LIN {X 0,Y 69.848,Z 476.675,A -85,B 0,C 180,E1 -28499.796,E2 -28499.796} C_VEL
LIN {X 0,Y 67.103,Z 478.987,A -85,B 0,C 180,E1 -28505.233,E2 -28505.233} C_VEL
LIN {X 0,Y 64.997,Z 480.714,A -85,B 0,C 180,E1 -28511.072,E2 -28511.072} C_VEL
LIN {X 0,Y 63.489,Z 481.949,A -85,B 0,C 180,E1 -28517.21,E2 -28517.21} C_VEL
LIN {X 0,Y 62.689,Z 482.712,A -85,B 0,C 180,E1 -28523.563,E2 -28523.563} C_VEL
LIN {X 0,Y 62.51,Z 483,A -85,B 0,C 180,E1 -28530,E2 -28530} C_VEL
LIN {X 0,Y 62.687,Z 482.698,A -85,B 0,C 180,E1 -28536.437,E2 -28536.437} C_VEL
LIN {X 0,Y 63.483,Z 481.907,A -85,B 0,C 180,E1 -28542.792,E2 -28542.792} C_VEL
LIN {X 0,Y 64.985,Z 480.644,A -85,B 0,C 180,E1 -28548.931,E2 -28548.931} C_VEL
LIN {X 0,Y 68.386,Z 477.737,A -85,B 0,C 180,E1 -28557.546,E2 -28557.546} C_VEL
LIN {X 0,Y 71.407,Z 475.084,A -85,B 0,C 180,E1 -28562.773,E2 -28562.773} C_VEL
LIN {X 0,Y 76.916,Z 469.904,A -85,B 0,C 180,E1 -28569.761,E2 -28569.761} C_VEL
LIN {X 0,Y 83.46,Z 463.065,A -85,B 0,C 180,E1 -28575.705,E2 -28575.705} C_VEL
LIN {X 0,Y 89.457,Z 455.594,A -85,B 0,C 180,E1 -28579.993,E2 -28579.993} C_VEL
LIN {X 0,Y 94.61,Z 448.222,A -85,B 0,C 180,E1 -28582.99,E2 -28582.99} C_VEL
LIN {X 0,Y 99.158,Z 440.542,A -85,B 0,C 180,E1 -28585.32,E2 -28585.32} C_VEL
LIN {X 0,Y 103.34,Z 431.965,A -85,B 0,C 180,E1 -28587.308,E2 -28587.308} C_VEL
LIN {X 0,Y 107.288,Z 421.966,A -85,B 0,C 180,E1 -28588.97,E2 -28588.97} C_VEL
LIN {X 0,Y 110.604,Z 410.25,A -85,B 0,C 180,E1 -28590.22,E2 -28590.22} C_VEL
LIN {X 0,Y 112.44,Z 400.537,A -85,B 0,C 180,E1 -28590.874,E2 -28590.874} C_VEL
LIN {X 0,Y 112.912,Z 396.513,A -85,B 0,C 180,E1 -28591.157,E2 -28591.157} C_VEL
LIN {X 0,Y 109.721,Z 389.352,A -85,B 0,C 180,E1 -28595.466,E2 -28595.466} C_VEL
LIN {X 0,Y 107.221,Z 384.494,A -85,B 0,C 180,E1 -28599.466,E2 -28599.466} C_VEL
LIN {X 0,Y 105.6,Z 381.525,A -85,B 0,C 180,E1 -28602.605,E2 -28602.605} C_VEL
LIN {X 0,Y 103.774,Z 378.179,A -85,B 0,C 180,E1 -28607.159,E2 -28607.159} C_VEL
LIN {X 0,Y 102.189,Z 375.125,A -85,B 0,C 180,E1 -28613.584,E2 -28613.584} C_VEL
LIN {X 0,Y 101.944,Z 373.871,A -85,B 0,C 180,E1 -28616.047,E2 -28616.047} C_VEL
LIN {X 0,Y 101.743,Z 373.505,A -85,B 0,C 180,E1 -28620,E2 -28620} C_VEL
LIN {X 0,Y 102.017,Z 374.037,A -85,B 0,C 180,E1 -28624.693,E2 -28624.693} C_VEL
LIN {X 0,Y 103.212,Z 377.51,A -85,B 0,C 180,E1 -28631.209,E2 -28631.209} C_VEL
LIN {X 0,Y 104.184,Z 378.885,A -85,B 0,C 180,E1 -28634.039,E2 -28634.039} C_VEL
LIN {X 0,Y 106.507,Z 383.167,A -85,B 0,C 180,E1 -28639.265,E2 -28639.265} C_VEL
LIN {X 0,Y 108.728,Z 387.363,A -85,B 0,C 180,E1 -28643.08,E2 -28643.08} C_VEL
LIN {X 0,Y 111.51,Z 393.241,A -85,B 0,C 180,E1 -28647.064,E2 -28647.064} C_VEL
LIN {X 0,Y 112.912,Z 396.627,A -85,B 0,C 180,E1 -28648.909,E2 -28648.909} C_VEL
LIN {X 0,Y 111.228,Z 407.408,A -85,B 0,C 180,E1 -28649.608,E2 -28649.608} C_VEL
LIN {X 0,Y 111.11,Z 407.875,A -85,B 0,C 180,E1 -28649.629,E2 -28649.629} C_VEL
LIN {X 0,Y 108.536,Z 415.532,A -85,B 0,C 180,E1 -28649.681,E2 -28649.681} C_VEL
LIN {X 0,Y 105.062,Z 422.853,A -85,B 0,C 180,E1 -28649.456,E2 -28649.456} C_VEL
LIN {X 0,Y 100.321,Z 431.414,A -85,B 0,C 180,E1 -28649.539,E2 -28649.539} C_VEL
LIN {X 0,Y 97.661,Z 436.251,A -85,B 0,C 180,E1 -28650.185,E2 -28650.185} C_VEL
LIN {X 0,Y 91.957,Z 446.132,A -85,B 0,C 180,E1 -28652.788,E2 -28652.788} C_VEL
LIN {X 0,Y 86.43,Z 453.852,A -85,B 0,C 180,E1 -28655.598,E2 -28655.598} C_VEL
LIN {X 0,Y 81.208,Z 460.199,A -85,B 0,C 180,E1 -28658.843,E2 -28658.843} C_VEL
LIN {X 0,Y 76.245,Z 465.475,A -85,B 0,C 180,E1 -28662.49,E2 -28662.49} C_VEL
LIN {X 0,Y 71.621,Z 469.88,A -85,B 0,C 180,E1 -28666.617,E2 -28666.617} C_VEL
LIN {X 0,Y 65.574,Z 475.065,A -85,B 0,C 180,E1 -28673.882,E2 -28673.882} C_VEL
LIN {X 0,Y 62.209,Z 477.722,A -85,B 0,C 180,E1 -28679.445,E2 -28679.445} C_VEL
LIN {X 0,Y 58.304,Z 480.634,A -85,B 0,C 180,E1 -28688.801,E2 -28688.801} C_VEL
LIN {X 0,Y 56.597,Z 481.901,A -85,B 0,C 180,E1 -28695.62,E2 -28695.62} C_VEL
LIN {X 0,Y 55.633,Z 482.696,A -85,B 0,C 180,E1 -28702.743,E2 -28702.743} C_VEL
LIN {X 0,Y 55.414,Z 482.999,A -85,B 0,C 180,E1 -28710,E2 -28710} C_VEL
LIN {X 0,Y 55.633,Z 482.714,A -85,B 0,C 180,E1 -28717.257,E2 -28717.257} C_VEL
LIN {X 0,Y 56.596,Z 481.955,A -85,B 0,C 180,E1 -28724.38,E2 -28724.38} C_VEL
LIN {X 0,Y 58.299,Z 480.725,A -85,B 0,C 180,E1 -28731.201,E2 -28731.201} C_VEL
LIN {X 0,Y 62.166,Z 477.851,A -85,B 0,C 180,E1 -28740.579,E2 -28740.579} C_VEL
LIN {X 0,Y 65.535,Z 475.234,A -85,B 0,C 180,E1 -28746.143,E2 -28746.143} C_VEL
LIN {X 0,Y 71.592,Z 470.095,A -85,B 0,C 180,E1 -28753.405,E2 -28753.405} C_VEL
LIN {X 0,Y 77.406,Z 464.567,A -85,B 0,C 180,E1 -28758.507,E2 -28758.507} C_VEL
LIN {X 0,Y 83.747,Z 457.615,A -85,B 0,C 180,E1 -28762.865,E2 -28762.865} C_VEL
LIN {X 0,Y 89.827,Z 449.637,A -85,B 0,C 180,E1 -28766.23,E2 -28766.23} C_VEL
LIN {X 0,Y 94.868,Z 441.786,A -85,B 0,C 180,E1 -28768.624,E2 -28768.624} C_VEL
LIN {X 0,Y 98.991,Z 434.053,A -85,B 0,C 180,E1 -28770.422,E2 -28770.422} C_VEL
LIN {X 0,Y 102.605,Z 425.802,A -85,B 0,C 180,E1 -28771.868,E2 -28771.868} C_VEL
LIN {X 0,Y 105.581,Z 417.212,A -85,B 0,C 180,E1 -28772.998,E2 -28772.998} C_VEL
LIN {X 0,Y 108.054,Z 407.867,A -85,B 0,C 180,E1 -28773.822,E2 -28773.822} C_VEL
LIN {X 0,Y 109.442,Z 400.033,A -85,B 0,C 180,E1 -28774.344,E2 -28774.344} C_VEL
LIN {X 0,Y 107.116,Z 394.028,A -85,B 0,C 180,E1 -28778.389,E2 -28778.389} C_VEL
LIN {X 0,Y 105.229,Z 390.11,A -85,B 0,C 180,E1 -28781.975,E2 -28781.975} C_VEL
LIN {X 0,Y 104.07,Z 387.868,A -85,B 0,C 180,E1 -28784.61,E2 -28784.61} C_VEL
LIN {X 0,Y 102.85,Z 385.178,A -85,B 0,C 180,E1 -28788.17,E2 -28788.17} C_VEL
LIN {X 0,Y 101.381,Z 381.825,A -85,B 0,C 180,E1 -28795.527,E2 -28795.527} C_VEL
LIN {X 0,Y 101.306,Z 381.029,A -85,B 0,C 180,E1 -28797.017,E2 -28797.017} C_VEL
LIN {X 0,Y 101.207,Z 380.698,A -85,B 0,C 180,E1 -28800,E2 -28800} C_VEL
LIN {X 0,Y 101.327,Z 381.227,A -85,B 0,C 180,E1 -28803.479,E2 -28803.479} C_VEL
LIN {X 0,Y 102.534,Z 384.8,A -85,B 0,C 180,E1 -28810.864,E2 -28810.864} C_VEL
LIN {X 0,Y 103.118,Z 385.874,A -85,B 0,C 180,E1 -28812.781,E2 -28812.781} C_VEL
LIN {X 0,Y 104.964,Z 389.588,A -85,B 0,C 180,E1 -28817.504,E2 -28817.504} C_VEL
LIN {X 0,Y 106.974,Z 393.735,A -85,B 0,C 180,E1 -28821.411,E2 -28821.411} C_VEL
LIN {X 0,Y 109.14,Z 399.137,A -85,B 0,C 180,E1 -28825.182,E2 -28825.182} C_VEL
LIN {X 0,Y 109.44,Z 400.029,A -85,B 0,C 180,E1 -28825.698,E2 -28825.698} C_VEL
LIN {X 0,Y 108.079,Z 407.829,A -85,B 0,C 180,E1 -28826.237,E2 -28826.237} C_VEL
LIN {X 0,Y 105.622,Z 417.18,A -85,B 0,C 180,E1 -28827.076,E2 -28827.076} C_VEL
LIN {X 0,Y 102.616,Z 425.721,A -85,B 0,C 180,E1 -28828.144,E2 -28828.144} C_VEL
LIN {X 0,Y 98.992,Z 433.988,A -85,B 0,C 180,E1 -28829.579,E2 -28829.579} C_VEL
LIN {X 0,Y 94.079,Z 443.081,A -85,B 0,C 180,E1 -28831.716,E2 -28831.716} C_VEL
LIN {X 0,Y 87.769,Z 452.48,A -85,B 0,C 180,E1 -28834.842,E2 -28834.842} C_VEL
LIN {X 0,Y 82.475,Z 459.063,A -85,B 0,C 180,E1 -28837.982,E2 -28837.982} C_VEL
LIN {X 0,Y 77.428,Z 464.54,A -85,B 0,C 180,E1 -28841.512,E2 -28841.512} C_VEL
LIN {X 0,Y 71.605,Z 470.073,A -85,B 0,C 180,E1 -28846.605,E2 -28846.605} C_VEL
LIN {X 0,Y 65.542,Z 475.216,A -85,B 0,C 180,E1 -28853.861,E2 -28853.861} C_VEL
LIN {X 0,Y 60.733,Z 478.988,A -85,B 0,C 180,E1 -28862.428,E2 -28862.428} C_VEL
LIN {X 0,Y 58.308,Z 480.715,A -85,B 0,C 180,E1 -28868.802,E2 -28868.802} C_VEL
LIN {X 0,Y 56.6,Z 481.949,A -85,B 0,C 180,E1 -28875.621,E2 -28875.621} C_VEL
LIN {X 0,Y 55.633,Z 482.712,A -85,B 0,C 180,E1 -28882.743,E2 -28882.743} C_VEL
LIN {X 0,Y 55.412,Z 483,A -85,B 0,C 180,E1 -28890,E2 -28890} C_VEL
LIN {X 0,Y 55.631,Z 482.698,A -85,B 0,C 180,E1 -28897.258,E2 -28897.258} C_VEL
LIN {X 0,Y 56.594,Z 481.906,A -85,B 0,C 180,E1 -28904.38,E2 -28904.38} C_VEL
LIN {X 0,Y 58.299,Z 480.644,A -85,B 0,C 180,E1 -28911.201,E2 -28911.201} C_VEL
LIN {X 0,Y 62.174,Z 477.736,A -85,B 0,C 180,E1 -28920.575,E2 -28920.575} C_VEL
LIN {X 0,Y 65.537,Z 475.083,A -85,B 0,C 180,E1 -28926.142,E2 -28926.142} C_VEL
LIN {X 0,Y 71.604,Z 469.903,A -85,B 0,C 180,E1 -28933.396,E2 -28933.396} C_VEL
LIN {X 0,Y 78.672,Z 463.063,A -85,B 0,C 180,E1 -28939.403,E2 -28939.403} C_VEL
LIN {X 0,Y 85.067,Z 455.591,A -85,B 0,C 180,E1 -28943.658,E2 -28943.658} C_VEL
LIN {X 0,Y 90.522,Z 448.219,A -85,B 0,C 180,E1 -28946.574,E2 -28946.574} C_VEL
LIN {X 0,Y 94.728,Z 441.531,A -85,B 0,C 180,E1 -28948.573,E2 -28948.573} C_VEL
LIN {X 0,Y 98.974,Z 433.461,A -85,B 0,C 180,E1 -28950.439,E2 -28950.439} C_VEL
LIN {X 0,Y 102.601,Z 425.063,A -85,B 0,C 180,E1 -28951.872,E2 -28951.872} C_VEL
LIN {X 0,Y 105.779,Z 415.77,A -85,B 0,C 180,E1 -28953,E2 -28953} C_VEL
LIN {X 0,Y 108.637,Z 404.172,A -85,B 0,C 180,E1 -28953.921,E2 -28953.921} C_VEL
LIN {X 0,Y 109.195,Z 399.767,A -85,B 0,C 180,E1 -28954.249,E2 -28954.249} C_VEL
LIN {X 0,Y 106.787,Z 393.629,A -85,B 0,C 180,E1 -28958.399,E2 -28958.399} C_VEL
LIN {X 0,Y 104.405,Z 388.609,A -85,B 0,C 180,E1 -28963.109,E2 -28963.109} C_VEL
LIN {X 0,Y 102.537,Z 384.948,A -85,B 0,C 180,E1 -28968.134,E2 -28968.134} C_VEL
LIN {X 0,Y 101.136,Z 381.751,A -85,B 0,C 180,E1 -28974.892,E2 -28974.892} C_VEL
LIN {X 0,Y 100.984,Z 380.826,A -85,B 0,C 180,E1 -28977.008,E2 -28977.008} C_VEL
LIN {X 0,Y 100.877,Z 380.562,A -85,B 0,C 180,E1 -28980,E2 -28980} C_VEL
LIN {X 0,Y 101.06,Z 381.043,A -85,B 0,C 180,E1 -28983.988,E2 -28983.988} C_VEL
LIN {X 0,Y 102.175,Z 384.511,A -85,B 0,C 180,E1 -28990.741,E2 -28990.741} C_VEL
LIN {X 0,Y 102.8,Z 385.479,A -85,B 0,C 180,E1 -28992.752,E2 -28992.752} C_VEL
LIN {X 0,Y 104.924,Z 389.79,A -85,B 0,C 180,E1 -28998.101,E2 -28998.101} C_VEL
LIN {X 0,Y 107.067,Z 394.284,A -85,B 0,C 180,E1 -29002.136,E2 -29002.136} C_VEL
LIN {X 0,Y 109.207,Z 399.783,A -85,B 0,C 180,E1 -29005.813,E2 -29005.813} C_VEL
LIN {X 0,Y 107.612,Z 408.645,A -85,B 0,C 180,E1 -29006.411,E2 -29006.411} C_VEL
LIN {X 0,Y 105.378,Z 417.076,A -85,B 0,C 180,E1 -29007.185,E2 -29007.185} C_VEL
LIN {X 0,Y 102.652,Z 424.982,A -85,B 0,C 180,E1 -29008.181,E2 -29008.181} C_VEL
LIN {X 0,Y 99.032,Z 433.395,A -85,B 0,C 180,E1 -29009.62,E2 -29009.62} C_VEL
LIN {X 0,Y 97.661,Z 436.251,A -85,B 0,C 180,E1 -29010.185,E2 -29010.185} C_VEL
LIN {X 0,Y 95.606,Z 439.629,A -85,B 0,C 180,E1 -29010.555,E2 -29010.555} C_VEL
LIN {X 0,Y 91.177,Z 444.743,A -85,B 0,C 180,E1 -29010.341,E2 -29010.341} C_VEL
LIN {X 0,Y 86.386,Z 449.514,A -85,B 0,C 180,E1 -29010.271,E2 -29010.271} C_VEL
LIN {X 0,Y 83.766,Z 452.347,A -85,B 0,C 180,E1 -29010.96,E2 -29010.96} C_VEL
LIN {X 0,Y 78.347,Z 458.784,A -85,B 0,C 180,E1 -29013.928,E2 -29013.928} C_VEL
LIN {X 0,Y 71.644,Z 465.477,A -85,B 0,C 180,E1 -29018.302,E2 -29018.302} C_VEL
LIN {X 0,Y 66.644,Z 469.882,A -85,B 0,C 180,E1 -29022.424,E2 -29022.424} C_VEL
LIN {X 0,Y 62.033,Z 473.55,A -85,B 0,C 180,E1 -29027.176,E2 -29027.176} C_VEL
LIN {X 0,Y 58.033,Z 476.55,A -85,B 0,C 180,E1 -29032.735,E2 -29032.735} C_VEL
LIN {X 0,Y 54.549,Z 478.874,A -85,B 0,C 180,E1 -29038.98,E2 -29038.98} C_VEL
LIN {X 0,Y 51.743,Z 480.635,A -85,B 0,C 180,E1 -29045.954,E2 -29045.954} C_VEL
LIN {X 0,Y 49.745,Z 481.901,A -85,B 0,C 180,E1 -29053.587,E2 -29053.587} C_VEL
LIN {X 0,Y 48.606,Z 482.696,A -85,B 0,C 180,E1 -29061.687,E2 -29061.687} C_VEL
LIN {X 0,Y 48.331,Z 482.999,A -85,B 0,C 180,E1 -29070,E2 -29070} C_VEL
LIN {X 0,Y 48.606,Z 482.714,A -85,B 0,C 180,E1 -29078.313,E2 -29078.313} C_VEL
LIN {X 0,Y 49.744,Z 481.954,A -85,B 0,C 180,E1 -29086.413,E2 -29086.413} C_VEL
LIN {X 0,Y 51.737,Z 480.724,A -85,B 0,C 180,E1 -29094.048,E2 -29094.048} C_VEL
LIN {X 0,Y 56.155,Z 477.85,A -85,B 0,C 180,E1 -29104.276,E2 -29104.276} C_VEL
LIN {X 0,Y 59.94,Z 475.232,A -85,B 0,C 180,E1 -29110.155,E2 -29110.155} C_VEL
LIN {X 0,Y 66.616,Z 470.093,A -85,B 0,C 180,E1 -29117.602,E2 -29117.602} C_VEL
LIN {X 0,Y 72.901,Z 464.565,A -85,B 0,C 180,E1 -29122.686,E2 -29122.686} C_VEL
LIN {X 0,Y 79.649,Z 457.612,A -85,B 0,C 180,E1 -29126.954,E2 -29126.954} C_VEL
LIN {X 0,Y 86.092,Z 449.634,A -85,B 0,C 180,E1 -29130.151,E2 -29130.151} C_VEL
LIN {X 0,Y 91.495,Z 441.57,A -85,B 0,C 180,E1 -29132.486,E2 -29132.486} C_VEL
LIN {X 0,Y 95.689,Z 434.048,A -85,B 0,C 180,E1 -29134.118,E2 -29134.118} C_VEL
LIN {X 0,Y 99.457,Z 425.796,A -85,B 0,C 180,E1 -29135.474,E2 -29135.474} C_VEL
LIN {X 0,Y 102.56,Z 417.204,A -85,B 0,C 180,E1 -29136.526,E2 -29136.526} C_VEL
LIN {X 0,Y 105.273,Z 407.266,A -85,B 0,C 180,E1 -29137.312,E2 -29137.312} C_VEL
LIN {X 0,Y 106.055,Z 403.255,A -85,B 0,C 180,E1 -29137.671,E2 -29137.671} C_VEL
LIN {X 0,Y 104.029,Z 397.63,A -85,B 0,C 180,E1 -29142.207,E2 -29142.207} C_VEL
LIN {X 0,Y 102.654,Z 394.473,A -85,B 0,C 180,E1 -29145.82,E2 -29145.82} C_VEL
LIN {X 0,Y 101.484,Z 391.783,A -85,B 0,C 180,E1 -29149.715,E2 -29149.715} C_VEL
LIN {X 0,Y 100.378,Z 387.966,A -85,B 0,C 180,E1 -29157.993,E2 -29157.993} C_VEL
LIN {X 0,Y 100.341,Z 387.756,A -85,B 0,C 180,E1 -29160,E2 -29160} C_VEL
LIN {X 0,Y 100.4,Z 388.202,A -85,B 0,C 180,E1 -29162.758,E2 -29162.758} C_VEL
LIN {X 0,Y 101.311,Z 391.527,A -85,B 0,C 180,E1 -29169.672,E2 -29169.672} C_VEL
LIN {X 0,Y 101.849,Z 392.623,A -85,B 0,C 180,E1 -29171.694,E2 -29171.694} C_VEL
LIN {X 0,Y 103.509,Z 396.376,A -85,B 0,C 180,E1 -29176.51,E2 -29176.51} C_VEL
LIN {X 0,Y 105.106,Z 400.548,A -85,B 0,C 180,E1 -29180.371,E2 -29180.371} C_VEL
LIN {X 0,Y 106.087,Z 403.434,A -85,B 0,C 180,E1 -29182.462,E2 -29182.462} C_VEL
LIN {X 0,Y 103.416,Z 414.573,A -85,B 0,C 180,E1 -29183.281,E2 -29183.281} C_VEL
LIN {X 0,Y 100.236,Z 423.854,A -85,B 0,C 180,E1 -29184.291,E2 -29184.291} C_VEL
LIN {X 0,Y 96.448,Z 432.492,A -85,B 0,C 180,E1 -29185.615,E2 -29185.615} C_VEL
LIN {X 0,Y 92.281,Z 440.213,A -85,B 0,C 180,E1 -29187.19,E2 -29187.19} C_VEL
LIN {X 0,Y 87.556,Z 447.554,A -85,B 0,C 180,E1 -29189.202,E2 -29189.202} C_VEL
LIN {X 0,Y 82.485,Z 454.187,A -85,B 0,C 180,E1 -29191.568,E2 -29191.568} C_VEL
LIN {X 0,Y 76.917,Z 460.484,A -85,B 0,C 180,E1 -29194.682,E2 -29194.682} C_VEL
LIN {X 0,Y 71.618,Z 465.714,A -85,B 0,C 180,E1 -29198.276,E2 -29198.276} C_VEL
LIN {X 0,Y 66.629,Z 470.074,A -85,B 0,C 180,E1 -29202.41,E2 -29202.41} C_VEL
LIN {X 0,Y 59.946,Z 475.217,A -85,B 0,C 180,E1 -29209.85,E2 -29209.85} C_VEL
LIN {X 0,Y 54.532,Z 478.989,A -85,B 0,C 180,E1 -29218.969,E2 -29218.969} C_VEL
LIN {X 0,Y 51.745,Z 480.716,A -85,B 0,C 180,E1 -29225.955,E2 -29225.955} C_VEL
LIN {X 0,Y 49.748,Z 481.949,A -85,B 0,C 180,E1 -29233.588,E2 -29233.588} C_VEL
LIN {X 0,Y 48.606,Z 482.713,A -85,B 0,C 180,E1 -29241.687,E2 -29241.687} C_VEL
LIN {X 0,Y 48.33,Z 483,A -85,B 0,C 180,E1 -29250,E2 -29250} C_VEL
LIN {X 0,Y 48.605,Z 482.698,A -85,B 0,C 180,E1 -29258.314,E2 -29258.314} C_VEL
LIN {X 0,Y 49.743,Z 481.906,A -85,B 0,C 180,E1 -29266.413,E2 -29266.413} C_VEL
LIN {X 0,Y 51.737,Z 480.643,A -85,B 0,C 180,E1 -29274.048,E2 -29274.048} C_VEL
LIN {X 0,Y 56.161,Z 477.735,A -85,B 0,C 180,E1 -29284.271,E2 -29284.271} C_VEL
LIN {X 0,Y 59.942,Z 475.082,A -85,B 0,C 180,E1 -29290.154,E2 -29290.154} C_VEL
LIN {X 0,Y 66.628,Z 469.901,A -85,B 0,C 180,E1 -29297.591,E2 -29297.591} C_VEL
LIN {X 0,Y 74.255,Z 463.06,A -85,B 0,C 180,E1 -29303.56,E2 -29303.56} C_VEL
LIN {X 0,Y 81.063,Z 455.589,A -85,B 0,C 180,E1 -29307.702,E2 -29307.702} C_VEL
LIN {X 0,Y 86.821,Z 448.216,A -85,B 0,C 180,E1 -29310.479,E2 -29310.479} C_VEL
LIN {X 0,Y 91.472,Z 441.122,A -85,B 0,C 180,E1 -29312.48,E2 -29312.48} C_VEL
LIN {X 0,Y 95.668,Z 433.456,A -85,B 0,C 180,E1 -29314.144,E2 -29314.144} C_VEL
LIN {X 0,Y 99.458,Z 425.058,A -85,B 0,C 180,E1 -29315.473,E2 -29315.473} C_VEL
LIN {X 0,Y 102.716,Z 415.898,A -85,B 0,C 180,E1 -29316.505,E2 -29316.505} C_VEL
LIN {X 0,Y 105.602,Z 404.687,A -85,B 0,C 180,E1 -29317.346,E2 -29317.346} C_VEL
LIN {X 0,Y 105.836,Z 403.192,A -85,B 0,C 180,E1 -29317.482,E2 -29317.482} C_VEL
LIN {X 0,Y 103.909,Z 397.7,A -85,B 0,C 180,E1 -29321.771,E2 -29321.771} C_VEL
LIN {X 0,Y 102.426,Z 394.324,A -85,B 0,C 180,E1 -29325.574,E2 -29325.574} C_VEL
LIN {X 0,Y 101.222,Z 391.613,A -85,B 0,C 180,E1 -29329.499,E2 -29329.499} C_VEL
LIN {X 0,Y 100.139,Z 388.355,A -85,B 0,C 180,E1 -29336.228,E2 -29336.228} C_VEL
LIN {X 0,Y 100.117,Z 387.894,A -85,B 0,C 180,E1 -29336.983,E2 -29336.983} C_VEL
LIN {X 0,Y 100.011,Z 387.615,A -85,B 0,C 180,E1 -29340,E2 -29340} C_VEL
LIN {X 0,Y 100.12,Z 388.037,A -85,B 0,C 180,E1 -29343.27,E2 -29343.27} C_VEL
LIN {X 0,Y 101.222,Z 391.625,A -85,B 0,C 180,E1 -29350.55,E2 -29350.55} C_VEL
LIN {X 0,Y 101.914,Z 393.301,A -85,B 0,C 180,E1 -29352.997,E2 -29352.997} C_VEL
LIN {X 0,Y 103.278,Z 396.24,A -85,B 0,C 180,E1 -29356.709,E2 -29356.709} C_VEL
LIN {X 0,Y 104.809,Z 400.186,A -85,B 0,C 180,E1 -29360.382,E2 -29360.382} C_VEL
LIN {X 0,Y 105.835,Z 403.175,A -85,B 0,C 180,E1 -29362.558,E2 -29362.558} C_VEL
LIN {X 0,Y 103.113,Z 414.619,A -85,B 0,C 180,E1 -29363.4,E2 -29363.4} C_VEL
LIN {X 0,Y 100.258,Z 423.116,A -85,B 0,C 180,E1 -29364.318,E2 -29364.318} C_VEL
LIN {X 0,Y 96.465,Z 431.9,A -85,B 0,C 180,E1 -29365.635,E2 -29365.635} C_VEL
LIN {X 0,Y 91.719,Z 440.758,A -85,B 0,C 180,E1 -29367.51,E2 -29367.51} C_VEL
LIN {X 0,Y 86.826,Z 448.177,A -85,B 0,C 180,E1 -29369.527,E2 -29369.527} C_VEL
LIN {X 0,Y 83.766,Z 452.347,A -85,B 0,C 180,E1 -29370.96,E2 -29370.96} C_VEL
LIN {X 0,Y 79.926,Z 456.561,A -85,B 0,C 180,E1 -29372.362,E2 -29372.362} C_VEL
LIN {X 0,Y 72.457,Z 462.764,A -85,B 0,C 180,E1 -29373.995,E2 -29373.995} C_VEL
LIN {X 0,Y 64.692,Z 468.201,A -85,B 0,C 180,E1 -29376.298,E2 -29376.298} C_VEL
LIN {X 0,Y 60.511,Z 471.045,A -85,B 0,C 180,E1 -29378.949,E2 -29378.949} C_VEL
LIN {X 0,Y 54.728,Z 475.068,A -85,B 0,C 180,E1 -29385.068,E2 -29385.068} C_VEL
LIN {X 0,Y 50.486,Z 477.724,A -85,B 0,C 180,E1 -29391.214,E2 -29391.214} C_VEL
LIN {X 0,Y 45.354,Z 480.635,A -85,B 0,C 180,E1 -29402.299,E2 -29402.299} C_VEL
LIN {X 0,Y 42.986,Z 481.901,A -85,B 0,C 180,E1 -29410.914,E2 -29410.914} C_VEL
LIN {X 0,Y 41.591,Z 482.697,A -85,B 0,C 180,E1 -29420.272,E2 -29420.272} C_VEL
LIN {X 0,Y 41.228,Z 482.999,A -85,B 0,C 180,E1 -29430,E2 -29430} C_VEL
LIN {X 0,Y 41.591,Z 482.714,A -85,B 0,C 180,E1 -29439.728,E2 -29439.728} C_VEL
LIN {X 0,Y 42.985,Z 481.954,A -85,B 0,C 180,E1 -29449.086,E2 -29449.086} C_VEL
LIN {X 0,Y 45.348,Z 480.724,A -85,B 0,C 180,E1 -29457.705,E2 -29457.705} C_VEL
LIN {X 0,Y 50.44,Z 477.849,A -85,B 0,C 180,E1 -29468.828,E2 -29468.828} C_VEL
LIN {X 0,Y 54.686,Z 475.231,A -85,B 0,C 180,E1 -29474.977,E2 -29474.977} C_VEL
LIN {X 0,Y 62.057,Z 470.092,A -85,B 0,C 180,E1 -29482.442,E2 -29482.442} C_VEL
LIN {X 0,Y 68.835,Z 464.563,A -85,B 0,C 180,E1 -29487.384,E2 -29487.384} C_VEL
LIN {X 0,Y 76.003,Z 457.61,A -85,B 0,C 180,E1 -29491.455,E2 -29491.455} C_VEL
LIN {X 0,Y 82.786,Z 449.63,A -85,B 0,C 180,E1 -29494.418,E2 -29494.418} C_VEL
LIN {X 0,Y 87.719,Z 442.709,A -85,B 0,C 180,E1 -29496.314,E2 -29496.314} C_VEL
LIN {X 0,Y 92.814,Z 434.044,A -85,B 0,C 180,E1 -29498.058,E2 -29498.058} C_VEL
LIN {X 0,Y 96.723,Z 425.79,A -85,B 0,C 180,E1 -29499.307,E2 -29499.307} C_VEL
LIN {X 0,Y 99.796,Z 417.647,A -85,B 0,C 180,E1 -29500.221,E2 -29500.221} C_VEL
LIN {X 0,Y 102.51,Z 408.215,A -85,B 0,C 180,E1 -29500.912,E2 -29500.912} C_VEL
LIN {X 0,Y 102.748,Z 406.686,A -85,B 0,C 180,E1 -29501.219,E2 -29501.219} C_VEL
LIN {X 0,Y 101.61,Z 402.59,A -85,B 0,C 180,E1 -29505.139,E2 -29505.139} C_VEL
LIN {X 0,Y 100.271,Z 398.668,A -85,B 0,C 180,E1 -29510.417,E2 -29510.417} C_VEL
LIN {X 0,Y 99.48,Z 394.896,A -85,B 0,C 180,E1 -29518.988,E2 -29518.988} C_VEL
LIN {X 0,Y 99.486,Z 395.21,A -85,B 0,C 180,E1 -29522.024,E2 -29522.024} C_VEL
LIN {X 0,Y 100.405,Z 399.148,A -85,B 0,C 180,E1 -29530.332,E2 -29530.332} C_VEL
LIN {X 0,Y 101.622,Z 402.66,A -85,B 0,C 180,E1 -29534.958,E2 -29534.958} C_VEL
LIN {X 0,Y 102.72,Z 406.524,A -85,B 0,C 180,E1 -29538.706,E2 -29538.706} C_VEL
LIN {X 0,Y 102.772,Z 407.166,A -85,B 0,C 180,E1 -29539.084,E2 -29539.084} C_VEL
LIN {X 0,Y 100.248,Z 416.327,A -85,B 0,C 180,E1 -29539.732,E2 -29539.732} C_VEL
LIN {X 0,Y 97.533,Z 423.86,A -85,B 0,C 180,E1 -29540.49,E2 -29540.49} C_VEL
LIN {X 0,Y 93.599,Z 432.497,A -85,B 0,C 180,E1 -29541.695,E2 -29541.695} C_VEL
LIN {X 0,Y 89.853,Z 439.269,A -85,B 0,C 180,E1 -29542.917,E2 -29542.917} C_VEL
LIN {X 0,Y 84.322,Z 447.557,A -85,B 0,C 180,E1 -29544.99,E2 -29544.99} C_VEL
LIN {X 0,Y 79.006,Z 454.189,A -85,B 0,C 180,E1 -29547.186,E2 -29547.186} C_VEL
LIN {X 0,Y 73.106,Z 460.486,A -85,B 0,C 180,E1 -29550.096,E2 -29550.096} C_VEL
LIN {X 0,Y 67.455,Z 465.716,A -85,B 0,C 180,E1 -29553.542,E2 -29553.542} C_VEL
LIN {X 0,Y 62.069,Z 470.076,A -85,B 0,C 180,E1 -29557.572,E2 -29557.572} C_VEL
LIN {X 0,Y 54.708,Z 475.218,A -85,B 0,C 180,E1 -29565.046,E2 -29565.046} C_VEL
LIN {X 0,Y 48.566,Z 478.99,A -85,B 0,C 180,E1 -29574.632,E2 -29574.632} C_VEL
LIN {X 0,Y 45.354,Z 480.716,A -85,B 0,C 180,E1 -29582.299,E2 -29582.299} C_VEL
LIN {X 0,Y 42.988,Z 481.95,A -85,B 0,C 180,E1 -29590.915,E2 -29590.915} C_VEL
LIN {X 0,Y 41.591,Z 482.713,A -85,B 0,C 180,E1 -29600.272,E2 -29600.272} C_VEL
LIN {X 0,Y 41.226,Z 483,A -85,B 0,C 180,E1 -29610,E2 -29610} C_VEL
LIN {X 0,Y 41.589,Z 482.698,A -85,B 0,C 180,E1 -29619.729,E2 -29619.729} C_VEL
LIN {X 0,Y 42.984,Z 481.906,A -85,B 0,C 180,E1 -29629.087,E2 -29629.087} C_VEL
LIN {X 0,Y 45.348,Z 480.642,A -85,B 0,C 180,E1 -29637.705,E2 -29637.705} C_VEL
LIN {X 0,Y 50.445,Z 477.734,A -85,B 0,C 180,E1 -29648.824,E2 -29648.824} C_VEL
LIN {X 0,Y 54.687,Z 475.081,A -85,B 0,C 180,E1 -29654.976,E2 -29654.976} C_VEL
LIN {X 0,Y 62.068,Z 469.9,A -85,B 0,C 180,E1 -29662.428,E2 -29662.428} C_VEL
LIN {X 0,Y 70.276,Z 463.058,A -85,B 0,C 180,E1 -29668.214,E2 -29668.214} C_VEL
LIN {X 0,Y 77.505,Z 455.586,A -85,B 0,C 180,E1 -29672.139,E2 -29672.139} C_VEL
LIN {X 0,Y 83.549,Z 448.213,A -85,B 0,C 180,E1 -29674.723,E2 -29674.723} C_VEL
LIN {X 0,Y 88.766,Z 440.569,A -85,B 0,C 180,E1 -29676.68,E2 -29676.68} C_VEL
LIN {X 0,Y 93.572,Z 431.951,A -85,B 0,C 180,E1 -29678.348,E2 -29678.348} C_VEL
LIN {X 0,Y 98.308,Z 421.258,A -85,B 0,C 180,E1 -29679.746,E2 -29679.746} C_VEL
LIN {X 0,Y 101.783,Z 409.987,A -85,B 0,C 180,E1 -29680.692,E2 -29680.692} C_VEL
LIN {X 0,Y 102.541,Z 406.592,A -85,B 0,C 180,E1 -29681.001,E2 -29681.001} C_VEL
LIN {X 0,Y 101.481,Z 402.771,A -85,B 0,C 180,E1 -29684.593,E2 -29684.593} C_VEL
LIN {X 0,Y 100.511,Z 400.151,A -85,B 0,C 180,E1 -29687.892,E2 -29687.892} C_VEL
LIN {X 0,Y 99.864,Z 398.197,A -85,B 0,C 180,E1 -29690.889,E2 -29690.889} C_VEL
LIN {X 0,Y 99.195,Z 395.062,A -85,B 0,C 180,E1 -29697.462,E2 -29697.462} C_VEL
LIN {X 0,Y 99.144,Z 394.67,A -85,B 0,C 180,E1 -29700,E2 -29700} C_VEL
LIN {X 0,Y 99.198,Z 395.174,A -85,B 0,C 180,E1 -29702.792,E2 -29702.792} C_VEL
LIN {X 0,Y 100.159,Z 398.954,A -85,B 0,C 180,E1 -29710.561,E2 -29710.561} C_VEL
LIN {X 0,Y 101.397,Z 402.517,A -85,B 0,C 180,E1 -29715.187,E2 -29715.187} C_VEL
LIN {X 0,Y 102.55,Z 406.626,A -85,B 0,C 180,E1 -29719.075,E2 -29719.075} C_VEL
LIN {X 0,Y 100.088,Z 415.898,A -85,B 0,C 180,E1 -29719.799,E2 -29719.799} C_VEL
LIN {X 0,Y 96.765,Z 424.994,A -85,B 0,C 180,E1 -29720.758,E2 -29720.758} C_VEL
LIN {X 0,Y 92.843,Z 433.405,A -85,B 0,C 180,E1 -29721.986,E2 -29721.986} C_VEL
LIN {X 0,Y 88.036,Z 441.764,A -85,B 0,C 180,E1 -29723.666,E2 -29723.666} C_VEL
LIN {X 0,Y 82.042,Z 450.222,A -85,B 0,C 180,E1 -29725.915,E2 -29725.915} C_VEL
LIN {X 0,Y 74.614,Z 458.786,A -85,B 0,C 180,E1 -29729.395,E2 -29729.395} C_VEL
LIN {X 0,Y 67.478,Z 465.479,A -85,B 0,C 180,E1 -29733.572,E2 -29733.572} C_VEL
LIN {X 0,Y 62.082,Z 469.883,A -85,B 0,C 180,E1 -29737.588,E2 -29737.588} C_VEL
LIN {X 0,Y 60.511,Z 471.045,A -85,B 0,C 180,E1 -29738.949,E2 -29738.949} C_VEL
LIN {X 0,Y 56.347,Z 473.738,A -85,B 0,C 180,E1 -29742.141,E2 -29742.141} C_VEL
LIN {X 0,Y 45.301,Z 478.565,A -85,B 0,C 180,E1 -29749.994,E2 -29749.994} C_VEL
LIN {X 0,Y 39.699,Z 480.525,A -85,B 0,C 180,E1 -29757.101,E2 -29757.101} C_VEL
LIN {X 0,Y 37.691,Z 481.247,A -85,B 0,C 180,E1 -29762.006,E2 -29762.006} C_VEL
LIN {X 0,Y 34.606,Z 482.697,A -85,B 0,C 180,E1 -29778.283,E2 -29778.283} C_VEL
LIN {X 0,Y 34.125,Z 482.999,A -85,B 0,C 180,E1 -29790,E2 -29790} C_VEL
LIN {X 0,Y 34.605,Z 482.714,A -85,B 0,C 180,E1 -29801.717,E2 -29801.717} C_VEL
LIN {X 0,Y 36.34,Z 481.954,A -85,B 0,C 180,E1 -29812.754,E2 -29812.754} C_VEL
LIN {X 0,Y 39.208,Z 480.723,A -85,B 0,C 180,E1 -29822.53,E2 -29822.53} C_VEL
LIN {X 0,Y 45.125,Z 477.848,A -85,B 0,C 180,E1 -29834.494,E2 -29834.494} C_VEL
LIN {X 0,Y 49.903,Z 475.23,A -85,B 0,C 180,E1 -29840.765,E2 -29840.765} C_VEL
LIN {X 0,Y 57.994,Z 470.09,A -85,B 0,C 180,E1 -29848.024,E2 -29848.024} C_VEL
LIN {X 0,Y 65.288,Z 464.561,A -85,B 0,C 180,E1 -29852.63,E2 -29852.63} C_VEL
LIN {X 0,Y 72.877,Z 457.607,A -85,B 0,C 180,E1 -29856.365,E2 -29856.365} C_VEL
LIN {X 0,Y 79.979,Z 449.627,A -85,B 0,C 180,E1 -29859.007,E2 -29859.007} C_VEL
LIN {X 0,Y 85.249,Z 442.494,A -85,B 0,C 180,E1 -29860.745,E2 -29860.745} C_VEL
LIN {X 0,Y 90.402,Z 434.039,A -85,B 0,C 180,E1 -29862.235,E2 -29862.235} C_VEL
LIN {X 0,Y 94.453,Z 425.784,A -85,B 0,C 180,E1 -29863.33,E2 -29863.33} C_VEL
LIN {X 0,Y 98.064,Z 416.341,A -85,B 0,C 180,E1 -29864.245,E2 -29864.245} C_VEL
LIN {X 0,Y 99.78,Z 410.635,A -85,B 0,C 180,E1 -29864.672,E2 -29864.672} C_VEL
LIN {X 0,Y 99.071,Z 407.311,A -85,B 0,C 180,E1 -29868.57,E2 -29868.57} C_VEL
LIN {X 0,Y 98.662,Z 405.227,A -85,B 0,C 180,E1 -29871.809,E2 -29871.809} C_VEL
LIN {X 0,Y 98.318,Z 401.996,A -85,B 0,C 180,E1 -29878.976,E2 -29878.976} C_VEL
LIN {X 0,Y 98.311,Z 402.051,A -85,B 0,C 180,E1 -29881.152,E2 -29881.152} C_VEL
LIN {X 0,Y 98.793,Z 405.984,A -85,B 0,C 180,E1 -29889.484,E2 -29889.484} C_VEL
LIN {X 0,Y 99.478,Z 409.214,A -85,B 0,C 180,E1 -29893.848,E2 -29893.848} C_VEL
LIN {X 0,Y 99.778,Z 410.63,A -85,B 0,C 180,E1 -29895.366,E2 -29895.366} C_VEL
LIN {X 0,Y 96.788,Z 420.187,A -85,B 0,C 180,E1 -29896.163,E2 -29896.163} C_VEL
LIN {X 0,Y 92.017,Z 431.001,A -85,B 0,C 180,E1 -29897.314,E2 -29897.314} C_VEL
LIN {X 0,Y 87.156,Z 439.547,A -85,B 0,C 180,E1 -29898.679,E2 -29898.679} C_VEL
LIN {X 0,Y 81.579,Z 447.56,A -85,B 0,C 180,E1 -29900.47,E2 -29900.47} C_VEL
LIN {X 0,Y 76.032,Z 454.192,A -85,B 0,C 180,E1 -29902.433,E2 -29902.433} C_VEL
LIN {X 0,Y 69.815,Z 460.488,A -85,B 0,C 180,E1 -29905.045,E2 -29905.045} C_VEL
LIN {X 0,Y 63.813,Z 465.718,A -85,B 0,C 180,E1 -29908.231,E2 -29908.231} C_VEL
LIN {X 0,Y 58.006,Z 470.077,A -85,B 0,C 180,E1 -29911.994,E2 -29911.994} C_VEL
LIN {X 0,Y 49.919,Z 475.219,A -85,B 0,C 180,E1 -29919.257,E2 -29919.257} C_VEL
LIN {X 0,Y 42.96,Z 478.991,A -85,B 0,C 180,E1 -29929.129,E2 -29929.129} C_VEL
LIN {X 0,Y 39.213,Z 480.717,A -85,B 0,C 180,E1 -29937.475,E2 -29937.475} C_VEL
LIN {X 0,Y 36.343,Z 481.95,A -85,B 0,C 180,E1 -29947.248,E2 -29947.248} C_VEL
LIN {X 0,Y 34.605,Z 482.713,A -85,B 0,C 180,E1 -29958.283,E2 -29958.283} C_VEL
LIN {X 0,Y 34.123,Z 482.999,A -85,B 0,C 180,E1 -29970,E2 -29970} C_VEL
LIN {X 0,Y 34.604,Z 482.698,A -85,B 0,C 180,E1 -29981.718,E2 -29981.718} C_VEL
LIN {X 0,Y 36.339,Z 481.905,A -85,B 0,C 180,E1 -29992.755,E2 -29992.755} C_VEL
LIN {X 0,Y 39.208,Z 480.642,A -85,B 0,C 180,E1 -30002.529,E2 -30002.529} C_VEL
LIN {X 0,Y 45.129,Z 477.733,A -85,B 0,C 180,E1 -30014.489,E2 -30014.489} C_VEL
LIN {X 0,Y 49.905,Z 475.08,A -85,B 0,C 180,E1 -30020.763,E2 -30020.763} C_VEL
LIN {X 0,Y 58.005,Z 469.898,A -85,B 0,C 180,E1 -30028.007,E2 -30028.007} C_VEL
LIN {X 0,Y 66.815,Z 463.056,A -85,B 0,C 180,E1 -30033.388,E2 -30033.388} C_VEL
LIN {X 0,Y 74.456,Z 455.583,A -85,B 0,C 180,E1 -30036.968,E2 -30036.968} C_VEL
LIN {X 0,Y 80.774,Z 448.21,A -85,B 0,C 180,E1 -30039.28,E2 -30039.28} C_VEL
LIN {X 0,Y 86.439,Z 440.204,A -85,B 0,C 180,E1 -30041.087,E2 -30041.087} C_VEL
LIN {X 0,Y 92,Z 430.445,A -85,B 0,C 180,E1 -30042.72,E2 -30042.72} C_VEL
LIN {X 0,Y 96.926,Z 418.856,A -85,B 0,C 180,E1 -30043.891,E2 -30043.891} C_VEL
LIN {X 0,Y 99.537,Z 410.418,A -85,B 0,C 180,E1 -30044.553,E2 -30044.553} C_VEL
LIN {X 0,Y 98.786,Z 406.959,A -85,B 0,C 180,E1 -30048.645,E2 -30048.645} C_VEL
LIN {X 0,Y 98.389,Z 404.95,A -85,B 0,C 180,E1 -30051.787,E2 -30051.787} C_VEL
LIN {X 0,Y 98.012,Z 401.778,A -85,B 0,C 180,E1 -30058.845,E2 -30058.845} C_VEL
LIN {X 0,Y 98.005,Z 401.974,A -85,B 0,C 180,E1 -30061.798,E2 -30061.798} C_VEL
LIN {X 0,Y 98.539,Z 405.76,A -85,B 0,C 180,E1 -30069.614,E2 -30069.614} C_VEL
LIN {X 0,Y 99.232,Z 408.986,A -85,B 0,C 180,E1 -30073.962,E2 -30073.962} C_VEL
LIN {X 0,Y 99.524,Z 410.392,A -85,B 0,C 180,E1 -30075.45,E2 -30075.45} C_VEL
LIN {X 0,Y 96.109,Z 421.17,A -85,B 0,C 180,E1 -30076.309,E2 -30076.309} C_VEL
LIN {X 0,Y 91.225,Z 431.909,A -85,B 0,C 180,E1 -30077.571,E2 -30077.571} C_VEL
LIN {X 0,Y 86.281,Z 440.453,A -85,B 0,C 180,E1 -30079.016,E2 -30079.016} C_VEL
LIN {X 0,Y 80.784,Z 448.183,A -85,B 0,C 180,E1 -30080.739,E2 -30080.739} C_VEL
LIN {X 0,Y 74.472,Z 455.561,A -85,B 0,C 180,E1 -30083.059,E2 -30083.059} C_VEL
LIN {X 0,Y 66.832,Z 463.037,A -85,B 0,C 180,E1 -30086.642,E2 -30086.642} C_VEL
LIN {X 0,Y 58.032,Z 469.885,A -85,B 0,C 180,E1 -30092.036,E2 -30092.036} C_VEL
LIN {X 0,Y 52.499,Z 473.552,A -85,B 0,C 180,E1 -30096.564,E2 -30096.564} C_VEL
LIN {X 0,Y 47.494,Z 476.552,A -85,B 0,C 180,E1 -30102.28,E2 -30102.28} C_VEL
LIN {X 0,Y 42.981,Z 478.876,A -85,B 0,C 180,E1 -30109.153,E2 -30109.153} C_VEL
LIN {X 0,Y 37.691,Z 481.247,A -85,B 0,C 180,E1 -30122.006,E2 -30122.006} C_VEL
LIN {X 0,Y 35.002,Z 482.227,A -85,B 0,C 180,E1 -30130.191,E2 -30130.191} C_VEL
LIN {X 0,Y 32.129,Z 482.776,A -85,B 0,C 180,E1 -30139.057,E2 -30139.057} C_VEL
LIN {X 0,Y 29.085,Z 482.966,A -85,B 0,C 180,E1 -30152.95,E2 -30152.95} C_VEL
LIN {X 0,Y 28.653,Z 482.482,A -85,B 0,C 180,E1 -30170.838,E2 -30170.838} C_VEL
LIN {X 0,Y 29.551,Z 482.051,A -85,B 0,C 180,E1 -30176.432,E2 -30176.432} C_VEL
LIN {X 0,Y 33.427,Z 480.722,A -85,B 0,C 180,E1 -30189.104,E2 -30189.104} C_VEL
LIN {X 0,Y 40.367,Z 477.847,A -85,B 0,C 180,E1 -30201.577,E2 -30201.577} C_VEL
LIN {X 0,Y 45.738,Z 475.229,A -85,B 0,C 180,E1 -30207.683,E2 -30207.683} C_VEL
LIN {X 0,Y 54.564,Z 470.089,A -85,B 0,C 180,E1 -30214.368,E2 -30214.368} C_VEL
LIN {X 0,Y 62.343,Z 464.56,A -85,B 0,C 180,E1 -30218.437,E2 -30218.437} C_VEL
LIN {X 0,Y 70.335,Z 457.605,A -85,B 0,C 180,E1 -30221.666,E2 -30221.666} C_VEL
LIN {X 0,Y 77.722,Z 449.624,A -85,B 0,C 180,E1 -30223.893,E2 -30223.893} C_VEL
LIN {X 0,Y 83.17,Z 442.507,A -85,B 0,C 180,E1 -30225.358,E2 -30225.358} C_VEL
LIN {X 0,Y 88.464,Z 434.089,A -85,B 0,C 180,E1 -30226.609,E2 -30226.609} C_VEL
LIN {X 0,Y 92.507,Z 426.131,A -85,B 0,C 180,E1 -30227.51,E2 -30227.51} C_VEL
LIN {X 0,Y 95.802,Z 417.991,A -85,B 0,C 180,E1 -30228.201,E2 -30228.201} C_VEL
LIN {X 0,Y 96.78,Z 415.2,A -85,B 0,C 180,E1 -30228.367,E2 -30228.367} C_VEL
LIN {X 0,Y 96.923,Z 414.635,A -85,B 0,C 180,E1 -30228.556,E2 -30228.556} C_VEL
LIN {X 0,Y 96.622,Z 411.696,A -85,B 0,C 180,E1 -30233.211,E2 -30233.211} C_VEL
LIN {X 0,Y 96.718,Z 408.752,A -85,B 0,C 180,E1 -30240,E2 -30240} C_VEL
LIN {X 0,Y 96.725,Z 412.432,A -85,B 0,C 180,E1 -30248.224,E2 -30248.224} C_VEL
LIN {X 0,Y 96.927,Z 414.618,A -85,B 0,C 180,E1 -30251.481,E2 -30251.481} C_VEL
LIN {X 0,Y 96.79,Z 415.192,A -85,B 0,C 180,E1 -30251.7,E2 -30251.7} C_VEL
LIN {X 0,Y 93.011,Z 424.994,A -85,B 0,C 180,E1 -30252.416,E2 -30252.416} C_VEL
LIN {X 0,Y 89.276,Z 432.597,A -85,B 0,C 180,E1 -30253.201,E2 -30253.201} C_VEL
LIN {X 0,Y 84.994,Z 439.78,A -85,B 0,C 180,E1 -30254.188,E2 -30254.188} C_VEL
LIN {X 0,Y 79.377,Z 447.563,A -85,B 0,C 180,E1 -30255.667,E2 -30255.667} C_VEL
LIN {X 0,Y 73.621,Z 454.195,A -85,B 0,C 180,E1 -30257.333,E2 -30257.333} C_VEL
LIN {X 0,Y 67.117,Z 460.491,A -85,B 0,C 180,E1 -30259.543,E2 -30259.543} C_VEL
LIN {X 0,Y 60.777,Z 465.72,A -85,B 0,C 180,E1 -30262.322,E2 -30262.322} C_VEL
LIN {X 0,Y 54.576,Z 470.079,A -85,B 0,C 180,E1 -30265.658,E2 -30265.658} C_VEL
LIN {X 0,Y 45.748,Z 475.221,A -85,B 0,C 180,E1 -30272.338,E2 -30272.338} C_VEL
LIN {X 0,Y 37.872,Z 478.992,A -85,B 0,C 180,E1 -30282.074,E2 -30282.074} C_VEL
LIN {X 0,Y 33.431,Z 480.718,A -85,B 0,C 180,E1 -30290.901,E2 -30290.901} C_VEL
LIN {X 0,Y 29.923,Z 481.95,A -85,B 0,C 180,E1 -30301.983,E2 -30301.983} C_VEL
LIN {X 0,Y 27.694,Z 482.713,A -85,B 0,C 180,E1 -30315.3,E2 -30315.3} C_VEL
LIN {X 0,Y 27.032,Z 482.999,A -85,B 0,C 180,E1 -30330,E2 -30330} C_VEL
LIN {X 0,Y 27.693,Z 482.698,A -85,B 0,C 180,E1 -30344.701,E2 -30344.701} C_VEL
LIN {X 0,Y 29.92,Z 481.905,A -85,B 0,C 180,E1 -30358.02,E2 -30358.02} C_VEL
LIN {X 0,Y 33.427,Z 480.641,A -85,B 0,C 180,E1 -30369.104,E2 -30369.104} C_VEL
LIN {X 0,Y 40.37,Z 477.732,A -85,B 0,C 180,E1 -30381.572,E2 -30381.572} C_VEL
LIN {X 0,Y 45.738,Z 475.078,A -85,B 0,C 180,E1 -30387.681,E2 -30387.681} C_VEL
LIN {X 0,Y 54.576,Z 469.897,A -85,B 0,C 180,E1 -30394.343,E2 -30394.343} C_VEL
LIN {X 0,Y 63.954,Z 463.054,A -85,B 0,C 180,E1 -30399.076,E2 -30399.076} C_VEL
LIN {X 0,Y 71.98,Z 455.581,A -85,B 0,C 180,E1 -30402.166,E2 -30402.166} C_VEL
LIN {X 0,Y 78.544,Z 448.206,A -85,B 0,C 180,E1 -30404.126,E2 -30404.126} C_VEL
LIN {X 0,Y 84.333,Z 440.307,A -85,B 0,C 180,E1 -30405.635,E2 -30405.635} C_VEL
LIN {X 0,Y 89.947,Z 430.806,A -85,B 0,C 180,E1 -30406.979,E2 -30406.979} C_VEL
LIN {X 0,Y 94.769,Z 420.067,A -85,B 0,C 180,E1 -30407.942,E2 -30407.942} C_VEL
LIN {X 0,Y 96.466,Z 415.228,A -85,B 0,C 180,E1 -30408.222,E2 -30408.222} C_VEL
LIN {X 0,Y 96.678,Z 414.164,A -85,B 0,C 180,E1 -30408.753,E2 -30408.753} C_VEL
LIN {X 0,Y 96.41,Z 411.605,A -85,B 0,C 180,E1 -30412.671,E2 -30412.671} C_VEL
LIN {X 0,Y 96.402,Z 408.651,A -85,B 0,C 180,E1 -30419.478,E2 -30419.478} C_VEL
LIN {X 0,Y 96.338,Z 408.969,A -85,B 0,C 180,E1 -30421.307,E2 -30421.307} C_VEL
LIN {X 0,Y 96.464,Z 412.26,A -85,B 0,C 180,E1 -30428.379,E2 -30428.379} C_VEL
LIN {X 0,Y 96.691,Z 414.333,A -85,B 0,C 180,E1 -30431.515,E2 -30431.515} C_VEL
LIN {X 0,Y 96.48,Z 415.146,A -85,B 0,C 180,E1 -30431.777,E2 -30431.777} C_VEL
LIN {X 0,Y 93.103,Z 424.081,A -85,B 0,C 180,E1 -30432.439,E2 -30432.439} C_VEL
LIN {X 0,Y 89.184,Z 432.198,A -85,B 0,C 180,E1 -30433.269,E2 -30433.269} C_VEL
LIN {X 0,Y 84.48,Z 440.098,A -85,B 0,C 180,E1 -30434.392,E2 -30434.392} C_VEL
LIN {X 0,Y 78.552,Z 448.187,A -85,B 0,C 180,E1 -30435.893,E2 -30435.893} C_VEL
LIN {X 0,Y 71.99,Z 455.564,A -85,B 0,C 180,E1 -30437.859,E2 -30437.859} C_VEL
LIN {X 0,Y 63.968,Z 463.04,A -85,B 0,C 180,E1 -30440.958,E2 -30440.958} C_VEL
LIN {X 0,Y 54.594,Z 469.886,A -85,B 0,C 180,E1 -30445.696,E2 -30445.696} C_VEL
LIN {X 0,Y 45.762,Z 475.07,A -85,B 0,C 180,E1 -30452.364,E2 -30452.364} C_VEL
LIN {X 0,Y 40.4,Z 477.726,A -85,B 0,C 180,E1 -30458.483,E2 -30458.483} C_VEL
LIN {X 0,Y 33.434,Z 480.636,A -85,B 0,C 180,E1 -30470.906,E2 -30470.906} C_VEL
LIN {X 0,Y 29.922,Z 481.902,A -85,B 0,C 180,E1 -30481.982,E2 -30481.982} C_VEL
LIN {X 0,Y 27.695,Z 482.697,A -85,B 0,C 180,E1 -30495.3,E2 -30495.3} C_VEL
LIN {X 0,Y 27.034,Z 482.999,A -85,B 0,C 180,E1 -30510,E2 -30510} C_VEL
LIN {X 0,Y 27.695,Z 482.714,A -85,B 0,C 180,E1 -30524.7,E2 -30524.7} C_VEL
LIN {X 0,Y 29.551,Z 482.051,A -85,B 0,C 180,E1 -30536.432,E2 -30536.432} C_VEL
LIN {X 0,Y 31.697,Z 481.224,A -85,B 0,C 180,E1 -30546.616,E2 -30546.616} C_VEL
LIN {X 0,Y 35.446,Z 479.067,A -85,B 0,C 180,E1 -30561.912,E2 -30561.912} C_VEL
LIN {X 0,Y 40.919,Z 476.092,A -85,B 0,C 180,E1 -30573.596,E2 -30573.596} C_VEL
LIN {X 0,Y 45.355,Z 473.769,A -85,B 0,C 180,E1 -30577.928,E2 -30577.928} C_VEL
LIN {X 0,Y 55.144,Z 468.074,A -85,B 0,C 180,E1 -30582.908,E2 -30582.908} C_VEL
LIN {X 0,Y 63.402,Z 461.921,A -85,B 0,C 180,E1 -30585.907,E2 -30585.907} C_VEL
LIN {X 0,Y 70.127,Z 455.912,A -85,B 0,C 180,E1 -30587.717,E2 -30587.717} C_VEL
LIN {X 0,Y 77.368,Z 448.045,A -85,B 0,C 180,E1 -30589.317,E2 -30589.317} C_VEL
LIN {X 0,Y 82.602,Z 441.151,A -85,B 0,C 180,E1 -30590.358,E2 -30590.358} C_VEL
LIN {X 0,Y 87.601,Z 433.198,A -85,B 0,C 180,E1 -30591.236,E2 -30591.236} C_VEL
LIN {X 0,Y 91.614,Z 425.303,A -85,B 0,C 180,E1 -30591.915,E2 -30591.915} C_VEL
LIN {X 0,Y 94.186,Z 419.081,A -85,B 0,C 180,E1 -30592.494,E2 -30592.494} C_VEL
LIN {X 0,Y 94.186,Z 417.576,A -85,B 0,C 180,E1 -30595.72,E2 -30595.72} C_VEL
LIN {X 0,Y 94.588,Z 415.74,A -85,B 0,C 180,E1 -30600,E2 -30600} C_VEL
LIN {X 0,Y 94.191,Z 418.83,A -85,B 0,C 180,E1 -30607.139,E2 -30607.139} C_VEL
LIN {X 0,Y 94.179,Z 419.07,A -85,B 0,C 180,E1 -30607.5,E2 -30607.5} C_VEL
LIN {X 0,Y 93.872,Z 420.095,A -85,B 0,C 180,E1 -30607.811,E2 -30607.811} C_VEL
LIN {X 0,Y 89.082,Z 430.581,A -85,B 0,C 180,E1 -30608.518,E2 -30608.518} C_VEL
LIN {X 0,Y 83.538,Z 439.784,A -85,B 0,C 180,E1 -30609.462,E2 -30609.462} C_VEL
LIN {X 0,Y 77.865,Z 447.439,A -85,B 0,C 180,E1 -30610.596,E2 -30610.596} C_VEL
LIN {X 0,Y 71.826,Z 454.197,A -85,B 0,C 180,E1 -30611.918,E2 -30611.918} C_VEL
LIN {X 0,Y 65.086,Z 460.493,A -85,B 0,C 180,E1 -30613.641,E2 -30613.641} C_VEL
LIN {X 0,Y 58.448,Z 465.722,A -85,B 0,C 180,E1 -30615.861,E2 -30615.861} C_VEL
LIN {X 0,Y 51.898,Z 470.08,A -85,B 0,C 180,E1 -30618.574,E2 -30618.574} C_VEL
LIN {X 0,Y 42.373,Z 475.222,A -85,B 0,C 180,E1 -30624.188,E2 -30624.188} C_VEL
LIN {X 0,Y 33.53,Z 478.992,A -85,B 0,C 180,E1 -30633.03,E2 -30633.03} C_VEL
LIN {X 0,Y 28.272,Z 480.718,A -85,B 0,C 180,E1 -30641.777,E2 -30641.777} C_VEL
LIN {X 0,Y 23.896,Z 481.951,A -85,B 0,C 180,E1 -30653.97,E2 -30653.97} C_VEL
LIN {X 0,Y 20.918,Z 482.713,A -85,B 0,C 180,E1 -30670.368,E2 -30670.368} C_VEL
LIN {X 0,Y 19.952,Z 482.999,A -85,B 0,C 180,E1 -30690,E2 -30690} C_VEL
LIN {X 0,Y 20.917,Z 482.698,A -85,B 0,C 180,E1 -30709.633,E2 -30709.633} C_VEL
LIN {X 0,Y 23.893,Z 481.905,A -85,B 0,C 180,E1 -30726.034,E2 -30726.034} C_VEL
LIN {X 0,Y 28.269,Z 480.641,A -85,B 0,C 180,E1 -30738.229,E2 -30738.229} C_VEL
LIN {X 0,Y 36.384,Z 477.732,A -85,B 0,C 180,E1 -30750.367,E2 -30750.367} C_VEL
LIN {X 0,Y 42.367,Z 475.077,A -85,B 0,C 180,E1 -30755.831,E2 -30755.831} C_VEL
LIN {X 0,Y 51.898,Z 469.895,A -85,B 0,C 180,E1 -30761.426,E2 -30761.426} C_VEL
LIN {X 0,Y 61.776,Z 463.052,A -85,B 0,C 180,E1 -30765.237,E2 -30765.237} C_VEL
LIN {X 0,Y 70.136,Z 455.578,A -85,B 0,C 180,E1 -30767.682,E2 -30767.682} C_VEL
LIN {X 0,Y 76.897,Z 448.216,A -85,B 0,C 180,E1 -30769.211,E2 -30769.211} C_VEL
LIN {X 0,Y 82.859,Z 440.303,A -85,B 0,C 180,E1 -30770.388,E2 -30770.388} C_VEL
LIN {X 0,Y 88.874,Z 430.346,A -85,B 0,C 180,E1 -30771.506,E2 -30771.506} C_VEL
LIN {X 0,Y 93.606,Z 419.894,A -85,B 0,C 180,E1 -30772.192,E2 -30772.192} C_VEL
LIN {X 0,Y 93.954,Z 418.761,A -85,B 0,C 180,E1 -30772.495,E2 -30772.495} C_VEL
LIN {X 0,Y 94.352,Z 415.435,A -85,B 0,C 180,E1 -30780,E2 -30780} C_VEL
LIN {X 0,Y 93.94,Z 418.576,A -85,B 0,C 180,E1 -30787.161,E2 -30787.161} C_VEL
LIN {X 0,Y 93.932,Z 418.805,A -85,B 0,C 180,E1 -30787.522,E2 -30787.522} C_VEL
LIN {X 0,Y 93.599,Z 419.913,A -85,B 0,C 180,E1 -30787.851,E2 -30787.851} C_VEL
LIN {X 0,Y 88.195,Z 431.559,A -85,B 0,C 180,E1 -30788.702,E2 -30788.702} C_VEL
LIN {X 0,Y 82.907,Z 440.236,A -85,B 0,C 180,E1 -30789.655,E2 -30789.655} C_VEL
LIN {X 0,Y 76.912,Z 448.19,A -85,B 0,C 180,E1 -30790.802,E2 -30790.802} C_VEL
LIN {X 0,Y 70.142,Z 455.566,A -85,B 0,C 180,E1 -30792.341,E2 -30792.341} C_VEL
LIN {X 0,Y 61.787,Z 463.042,A -85,B 0,C 180,E1 -30794.801,E2 -30794.801} C_VEL
LIN {X 0,Y 51.91,Z 469.888,A -85,B 0,C 180,E1 -30798.614,E2 -30798.614} C_VEL
LIN {X 0,Y 42.383,Z 475.071,A -85,B 0,C 180,E1 -30804.216,E2 -30804.216} C_VEL
LIN {X 0,Y 36.408,Z 477.727,A -85,B 0,C 180,E1 -30809.699,E2 -30809.699} C_VEL
LIN {X 0,Y 28.276,Z 480.637,A -85,B 0,C 180,E1 -30821.786,E2 -30821.786} C_VEL
LIN {X 0,Y 23.896,Z 481.902,A -85,B 0,C 180,E1 -30833.97,E2 -30833.97} C_VEL
LIN {X 0,Y 20.918,Z 482.697,A -85,B 0,C 180,E1 -30850.369,E2 -30850.369} C_VEL
LIN {X 0,Y 19.954,Z 482.999,A -85,B 0,C 180,E1 -30870,E2 -30870} C_VEL
LIN {X 0,Y 20.918,Z 482.714,A -85,B 0,C 180,E1 -30889.632,E2 -30889.632} C_VEL
LIN {X 0,Y 23.894,Z 481.953,A -85,B 0,C 180,E1 -30906.033,E2 -30906.033} C_VEL
LIN {X 0,Y 28.269,Z 480.722,A -85,B 0,C 180,E1 -30918.23,E2 -30918.23} C_VEL
LIN {X 0,Y 36.382,Z 477.846,A -85,B 0,C 180,E1 -30930.373,E2 -30930.373} C_VEL
LIN {X 0,Y 42.366,Z 475.228,A -85,B 0,C 180,E1 -30935.833,E2 -30935.833} C_VEL
LIN {X 0,Y 45.355,Z 473.769,A -85,B 0,C 180,E1 -30937.928,E2 -30937.928} C_VEL
LIN {X 0,Y 49.913,Z 471.301,A -85,B 0,C 180,E1 -30941.409,E2 -30941.409} C_VEL
LIN {X 0,Y 56.73,Z 466.659,A -85,B 0,C 180,E1 -30947.418,E2 -30947.418} C_VEL
LIN {X 0,Y 63.46,Z 461.105,A -85,B 0,C 180,E1 -30951.935,E2 -30951.935} C_VEL
LIN {X 0,Y 67.636,Z 457.21,A -85,B 0,C 180,E1 -30953.27,E2 -30953.27} C_VEL
LIN {X 0,Y 74.685,Z 450.029,A -85,B 0,C 180,E1 -30954.306,E2 -30954.306} C_VEL
LIN {X 0,Y 81.103,Z 442.012,A -85,B 0,C 180,E1 -30955.183,E2 -30955.183} C_VEL
LIN {X 0,Y 86.013,Z 434.553,A -85,B 0,C 180,E1 -30955.798,E2 -30955.798} C_VEL
LIN {X 0,Y 90.558,Z 426.005,A -85,B 0,C 180,E1 -30956.32,E2 -30956.32} C_VEL
LIN {X 0,Y 91.049,Z 424.949,A -85,B 0,C 180,E1 -30956.374,E2 -30956.374} C_VEL
LIN {X 0,Y 91.504,Z 423.893,A -85,B 0,C 180,E1 -30956.806,E2 -30956.806} C_VEL
LIN {X 0,Y 91.96,Z 422.613,A -85,B 0,C 180,E1 -30960,E2 -30960} C_VEL
LIN {X 0,Y 91.504,Z 423.884,A -85,B 0,C 180,E1 -30963.193,E2 -30963.193} C_VEL
LIN {X 0,Y 91.052,Z 424.94,A -85,B 0,C 180,E1 -30963.659,E2 -30963.659} C_VEL
LIN {X 0,Y 86.83,Z 433.136,A -85,B 0,C 180,E1 -30964.117,E2 -30964.117} C_VEL
LIN {X 0,Y 81.97,Z 440.775,A -85,B 0,C 180,E1 -30964.687,E2 -30964.687} C_VEL
LIN {X 0,Y 76.174,Z 448.273,A -85,B 0,C 180,E1 -30965.508,E2 -30965.508} C_VEL
LIN {X 0,Y 68.973,Z 455.904,A -85,B 0,C 180,E1 -30966.559,E2 -30966.559} C_VEL
LIN {X 0,Y 60.357,Z 463.32,A -85,B 0,C 180,E1 -30968.221,E2 -30968.221} C_VEL
LIN {X 0,Y 51.792,Z 469.126,A -85,B 0,C 180,E1 -30970.335,E2 -30970.335} C_VEL
LIN {X 0,Y 43.323,Z 473.706,A -85,B 0,C 180,E1 -30973.267,E2 -30973.267} C_VEL
LIN {X 0,Y 36.684,Z 476.682,A -85,B 0,C 180,E1 -30976.686,E2 -30976.686} C_VEL
LIN {X 0,Y 30.254,Z 478.993,A -85,B 0,C 180,E1 -30981.691,E2 -30981.691} C_VEL
LIN {X 0,Y 24.13,Z 480.719,A -85,B 0,C 180,E1 -30989.101,E2 -30989.101} C_VEL
LIN {X 0,Y 18.618,Z 481.951,A -85,B 0,C 180,E1 -31000.979,E2 -31000.979} C_VEL
LIN {X 0,Y 14.426,Z 482.713,A -85,B 0,C 180,E1 -31020.846,E2 -31020.846} C_VEL
LIN {X 0,Y 12.86,Z 482.999,A -85,B 0,C 180,E1 -31050,E2 -31050} C_VEL
LIN {X 0,Y 14.425,Z 482.698,A -85,B 0,C 180,E1 -31079.156,E2 -31079.156} C_VEL
LIN {X 0,Y 18.616,Z 481.904,A -85,B 0,C 180,E1 -31099.029,E2 -31099.029} C_VEL
LIN {X 0,Y 24.128,Z 480.64,A -85,B 0,C 180,E1 -31110.906,E2 -31110.906} C_VEL
LIN {X 0,Y 33.439,Z 477.731,A -85,B 0,C 180,E1 -31121.041,E2 -31121.041} C_VEL
LIN {X 0,Y 39.988,Z 475.076,A -85,B 0,C 180,E1 -31125.154,E2 -31125.154} C_VEL
LIN {X 0,Y 50.09,Z 469.894,A -85,B 0,C 180,E1 -31129.15,E2 -31129.15} C_VEL
LIN {X 0,Y 60.356,Z 463.049,A -85,B 0,C 180,E1 -31131.785,E2 -31131.785} C_VEL
LIN {X 0,Y 68.973,Z 455.575,A -85,B 0,C 180,E1 -31133.438,E2 -31133.438} C_VEL
LIN {X 0,Y 75.93,Z 448.165,A -85,B 0,C 180,E1 -31134.491,E2 -31134.491} C_VEL
LIN {X 0,Y 81.973,Z 440.299,A -85,B 0,C 180,E1 -31135.285,E2 -31135.285} C_VEL
LIN {X 0,Y 87.755,Z 430.949,A -85,B 0,C 180,E1 -31136.031,E2 -31136.031} C_VEL
LIN {X 0,Y 90.411,Z 425.581,A -85,B 0,C 180,E1 -31136.309,E2 -31136.309} C_VEL
LIN {X 0,Y 91.257,Z 423.692,A -85,B 0,C 180,E1 -31136.745,E2 -31136.745} C_VEL
LIN {X 0,Y 91.742,Z 422.341,A -85,B 0,C 180,E1 -31140,E2 -31140} C_VEL
LIN {X 0,Y 91.283,Z 423.639,A -85,B 0,C 180,E1 -31143.313,E2 -31143.313} C_VEL
LIN {X 0,Y 90.866,Z 424.607,A -85,B 0,C 180,E1 -31143.705,E2 -31143.705} C_VEL
LIN {X 0,Y 86.703,Z 432.769,A -85,B 0,C 180,E1 -31144.161,E2 -31144.161} C_VEL
LIN {X 0,Y 81.98,Z 440.292,A -85,B 0,C 180,E1 -31144.775,E2 -31144.775} C_VEL
LIN {X 0,Y 76.196,Z 447.848,A -85,B 0,C 180,E1 -31145.491,E2 -31145.491} C_VEL
LIN {X 0,Y 70.706,Z 453.868,A -85,B 0,C 180,E1 -31146.306,E2 -31146.306} C_VEL
LIN {X 0,Y 63.796,Z 460.212,A -85,B 0,C 180,E1 -31147.496,E2 -31147.496} C_VEL
LIN {X 0,Y 56.928,Z 465.486,A -85,B 0,C 180,E1 -31149.026,E2 -31149.026} C_VEL
LIN {X 0,Y 50.098,Z 469.89,A -85,B 0,C 180,E1 -31150.894,E2 -31150.894} C_VEL
LIN {X 0,Y 39.997,Z 475.073,A -85,B 0,C 180,E1 -31154.893,E2 -31154.893} C_VEL
LIN {X 0,Y 33.463,Z 477.728,A -85,B 0,C 180,E1 -31159.077,E2 -31159.077} C_VEL
LIN {X 0,Y 24.133,Z 480.638,A -85,B 0,C 180,E1 -31169.115,E2 -31169.115} C_VEL
LIN {X 0,Y 18.618,Z 481.903,A -85,B 0,C 180,E1 -31180.979,E2 -31180.979} C_VEL
LIN {X 0,Y 14.427,Z 482.697,A -85,B 0,C 180,E1 -31200.847,E2 -31200.847} C_VEL
LIN {X 0,Y 12.861,Z 482.999,A -85,B 0,C 180,E1 -31230,E2 -31230} C_VEL
LIN {X 0,Y 14.426,Z 482.714,A -85,B 0,C 180,E1 -31259.154,E2 -31259.154} C_VEL
LIN {X 0,Y 18.616,Z 481.953,A -85,B 0,C 180,E1 -31279.027,E2 -31279.027} C_VEL
LIN {X 0,Y 24.127,Z 480.721,A -85,B 0,C 180,E1 -31290.908,E2 -31290.908} C_VEL
LIN {X 0,Y 33.438,Z 477.845,A -85,B 0,C 180,E1 -31301.048,E2 -31301.048} C_VEL
LIN {X 0,Y 42.691,Z 473.995,A -85,B 0,C 180,E1 -31306.465,E2 -31306.465} C_VEL
LIN {X 0,Y 53.491,Z 468.072,A -85,B 0,C 180,E1 -31310.19,E2 -31310.19} C_VEL
LIN {X 0,Y 62.055,Z 461.919,A -85,B 0,C 180,E1 -31312.287,E2 -31312.287} C_VEL
LIN {X 0,Y 67.636,Z 457.21,A -85,B 0,C 180,E1 -31313.27,E2 -31313.27} C_VEL
LIN {X 0,Y 67.4,Z 457.339,A -85,B 0,C 180,E1 -31314.102,E2 -31314.102} C_VEL
LIN {X 0,Y 66.177,Z 458.321,A -85,B 0,C 180,E1 -31315.157,E2 -31315.157} C_VEL
LIN {X 0,Y 60.225,Z 462.972,A -85,B 0,C 180,E1 -31317.966,E2 -31317.966} C_VEL
LIN {X 0,Y 50.084,Z 469.645,A -85,B 0,C 180,E1 -31321.76,E2 -31321.76} C_VEL
LIN {X 0,Y 42.824,Z 473.432,A -85,B 0,C 180,E1 -31323.763,E2 -31323.763} C_VEL
LIN {X 0,Y 35.305,Z 476.683,A -85,B 0,C 180,E1 -31325.551,E2 -31325.551} C_VEL
LIN {X 0,Y 28.404,Z 478.994,A -85,B 0,C 180,E1 -31328.233,E2 -31328.233} C_VEL
LIN {X 0,Y 21.589,Z 480.719,A -85,B 0,C 180,E1 -31332.418,E2 -31332.418} C_VEL
LIN {X 0,Y 14.953,Z 481.952,A -85,B 0,C 180,E1 -31339.955,E2 -31339.955} C_VEL
LIN {X 0,Y 8.927,Z 482.713,A -85,B 0,C 180,E1 -31358.071,E2 -31358.071} C_VEL
LIN {X 0,Y 5.759,Z 482.999,A -85,B 0,C 180,E1 -31410,E2 -31410} C_VEL
LIN {X 0,Y 8.926,Z 482.697,A -85,B 0,C 180,E1 -31461.935,E2 -31461.935} C_VEL
LIN {X 0,Y 14.952,Z 481.904,A -85,B 0,C 180,E1 -31480.056,E2 -31480.056} C_VEL
LIN {X 0,Y 21.588,Z 480.639,A -85,B 0,C 180,E1 -31487.59,E2 -31487.59} C_VEL
LIN {X 0,Y 31.846,Z 477.73,A -85,B 0,C 180,E1 -31493.245,E2 -31493.245} C_VEL
LIN {X 0,Y 38.781,Z 475.075,A -85,B 0,C 180,E1 -31495.341,E2 -31495.341} C_VEL
LIN {X 0,Y 49.25,Z 469.892,A -85,B 0,C 180,E1 -31497.291,E2 -31497.291} C_VEL
LIN {X 0,Y 59.756,Z 463.047,A -85,B 0,C 180,E1 -31498.555,E2 -31498.555} C_VEL
LIN {X 0,Y 68.526,Z 455.572,A -85,B 0,C 180,E1 -31499.334,E2 -31499.334} C_VEL
LIN {X 0,Y 74.869,Z 448.988,A -85,B 0,C 180,E1 -31499.8,E2 -31499.8} C_VEL
LIN {X 0,Y 77.661,Z 445.742,A -85,B 0,C 180,E1 -31500.001,E2 -31500.001} C_VEL
LIN {X 0,Y 70.282,Z 453.871,A -85,B 0,C 180,E1 -31500.547,E2 -31500.547} C_VEL
LIN {X 0,Y 63.262,Z 460.215,A -85,B 0,C 180,E1 -31501.11,E2 -31501.11} C_VEL
LIN {X 0,Y 56.252,Z 465.488,A -85,B 0,C 180,E1 -31501.857,E2 -31501.857} C_VEL
LIN {X 0,Y 49.252,Z 469.891,A -85,B 0,C 180,E1 -31502.752,E2 -31502.752} C_VEL
LIN {X 0,Y 38.784,Z 475.074,A -85,B 0,C 180,E1 -31504.705,E2 -31504.705} C_VEL
LIN {X 0,Y 31.854,Z 477.729,A -85,B 0,C 180,E1 -31506.871,E2 -31506.871} C_VEL
LIN {X 0,Y 21.59,Z 480.638,A -85,B 0,C 180,E1 -31512.439,E2 -31512.439} C_VEL
LIN {X 0,Y 14.954,Z 481.903,A -85,B 0,C 180,E1 -31519.957,E2 -31519.957} C_VEL
LIN {X 0,Y 8.928,Z 482.697,A -85,B 0,C 180,E1 -31538.075,E2 -31538.075} C_VEL
LIN {X 0,Y 5.76,Z 482.999,A -85,B 0,C 180,E1 -31590,E2 -31590} C_VEL
LIN {X 0,Y 8.927,Z 482.714,A -85,B 0,C 180,E1 -31641.927,E2 -31641.927} C_VEL
LIN {X 0,Y 14.953,Z 481.952,A -85,B 0,C 180,E1 -31660.053,E2 -31660.053} C_VEL
LIN {X 0,Y 21.588,Z 480.72,A -85,B 0,C 180,E1 -31667.592,E2 -31667.592} C_VEL
LIN {X 0,Y 31.846,Z 477.844,A -85,B 0,C 180,E1 -31673.251,E2 -31673.251} C_VEL
LIN {X 0,Y 38.781,Z 475.225,A -85,B 0,C 180,E1 -31675.345,E2 -31675.345} C_VEL
LIN {X 0,Y 49.248,Z 470.084,A -85,B 0,C 180,E1 -31677.339,E2 -31677.339} C_VEL
LIN {X 0,Y 58.001,Z 464.554,A -85,B 0,C 180,E1 -31678.435,E2 -31678.435} C_VEL
LIN {X 0,Y 66.911,Z 457.461,A -85,B 0,C 180,E1 -31679.263,E2 -31679.263} C_VEL
LIN {X 0,Y 74.756,Z 449.515,A -85,B 0,C 180,E1 -31679.798,E2 -31679.798} C_VEL
LIN {X 0,Y 77.306,Z 446.552,A -85,B 0,C 180,E1 -31679.999,E2 -31679.999} C_VEL
LIN {X 0,Y 70.281,Z 454.203,A -85,B 0,C 180,E1 -31680.53,E2 -31680.53} C_VEL
LIN {X 0,Y 63.261,Z 460.497,A -85,B 0,C 180,E1 -31681.046,E2 -31681.046} C_VEL
LIN {X 0,Y 56.25,Z 465.725,A -85,B 0,C 180,E1 -31681.793,E2 -31681.793} C_VEL
LIN {X 0,Y 49.25,Z 470.083,A -85,B 0,C 180,E1 -31682.709,E2 -31682.709} C_VEL
LIN {X 0,Y 42.824,Z 473.432,A -85,B 0,C 180,E1 -31683.763,E2 -31683.763} C_VEL
LIN {X 0,Y 41.709,Z 475.23,A -85,B 0,C 180,E1 -31683.968,E2 -31683.968} C_VEL
LIN {X 0,Y 41.709,Z 600,A -85,B 0,C 180,E1 -31683.968,E2 -31683.968} C_VEL
LIN {X 0,Y 41.709,Z 600,A -85,B 0,C 180,E1 -31683.968,E2 -31683.968}

QRS_NEXT_CUT()

QRS_NEXT()
QRS_HOME()

END
